Staubli VAL3: saveIt.pgx

program saveIt(bool& x_bSave[])
  local string l_sMessage
  local num l_nResult
  local string l_sEmpty
begin
  // save
  x_bSave=false
  logMsg("[KERNEL] INTERFACE:Save the trajectory "+saveData:sTrajTypeUsing+": "+sPalletName)
  call language:message(l_sMessage,-4)
  call use:timerDialog(l_sMessage,1)
  call pallet:setPalletData(tTrajPallet)
  call pallet:onSave(l_sEmpty)
end
